{attribute 'qualified_only'}
{attribute 'strict'}
TYPE E_COE_PTP_TRANSPORT_LAYER :
(
	UNKNOWN := -1,
	PTP_OVER_ETHERNET := 0,
	PTP_OVER_UDP := 1
);
END_TYPE

(* stored: Version 1.1.0.1, ProductVersion 3.1.4022.12
   DUT E_COE_PTP_TRANSPORT_LAYER: Id {6b1bab8c-e7aa-4cb3-92ca-7eed67ffb775} *)
